{attribute 'enable_dynamic_creation'}
TYPE T_HashInfo :
STRUCT
	strBarcode	: STRING;
END_STRUCT
END_TYPE

(* stored: Version 1.1.0.1, ProductVersion 3.1.0.25
   DUT T_HashInfo: Id {6982fb26-dc01-46e0-be3f-6311c9ca8e06} *)
